// Mitsubishi GX Works2 project: plc0806   PLC: Q03UDV

PROGRAM MAIN
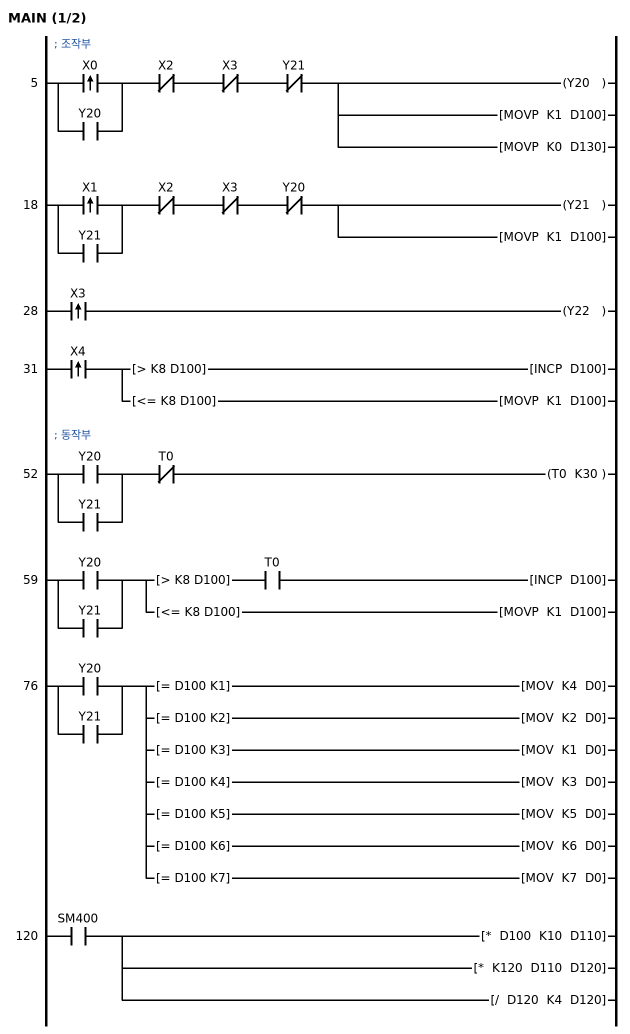
; 조작부
5     LDP     X0
      OR      Y20
      ANI     X2
      ANI     X3
      ANI     Y21
      OUT     Y20
      MOVP    K1 D100
      MOVP    K0 D130
18    LDP     X1
      OR      Y21
      ANI     X2
      ANI     X3
      ANI     Y20
      OUT     Y21
      MOVP    K1 D100
28    LDP     X3
      OUT     Y22
31    LDP     X4
      MPS
      AND>    K8 D100
      INCP    D100
      MPP
      AND<=   K8 D100
      MOVP    K1 D100
; 동작부
52    LD      Y20
      OR      Y21
      ANI     T0
      OUT     T0 K30
59    LD      Y20
      OR      Y21
      MPS
      AND>    K8 D100
      AND     T0
      INCP    D100
      MPP
      AND<=   K8 D100
      MOVP    K1 D100
76    LD      Y20
      OR      Y21
      MPS
      AND=    D100 K1
      MOV     K4 D0
      MRD
      AND=    D100 K2
      MOV     K2 D0
      MRD
      AND=    D100 K3
      MOV     K1 D0
      MRD
      AND=    D100 K4
      MOV     K3 D0
      MRD
      AND=    D100 K5
      MOV     K5 D0
      MRD
      AND=    D100 K6
      MOV     K6 D0
      MPP
      AND=    D100 K7
      MOV     K7 D0
120   LD      SM400
      *       D100 K10 D110
      *       K120 D110 D120
      /       D120 K4 D120
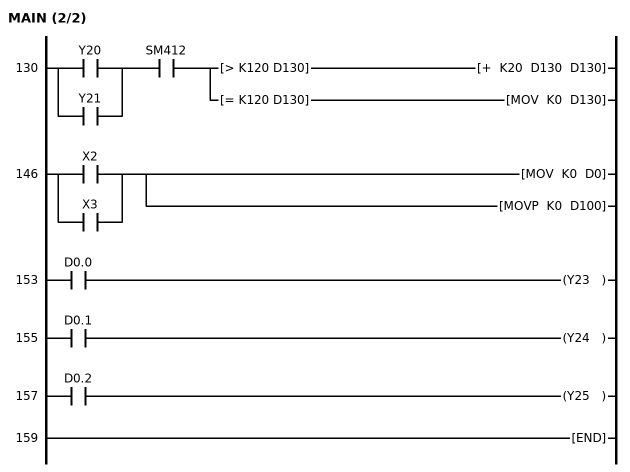
130   LD      Y20
      OR      Y21
      AND     SM412
      MPS
      AND>    K120 D130
      +       K20 D130 D130
      MPP
      AND=    K120 D130
      MOV     K0 D130
146   LD      X2
      OR      X3
      MOV     K0 D0
      MOVP    K0 D100
153   LD      D0.0
      OUT     Y23
155   LD      D0.1
      OUT     Y24
157   LD      D0.2
      OUT     Y25
159   END
END_PROGRAM

PROGRAM laundry
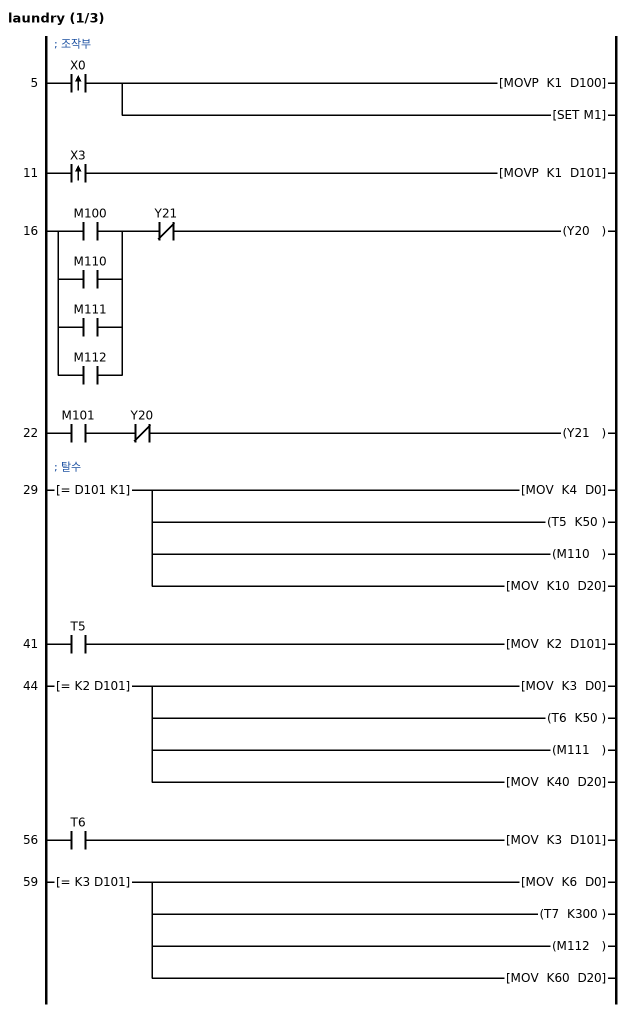
; 조작부
5     LDP     X0
      MOVP    K1 D100
      SET     M1
11    LDP     X3
      MOVP    K1 D101
16    LD      M100
      OR      M110
      OR      M111
      OR      M112
      ANI     Y21
      OUT     Y20
22    LD      M101
      ANI     Y20
      OUT     Y21
; 탈수
29    LD=     D101 K1
      MOV     K4 D0
      OUT     T5 K50
      OUT     M110
      MOV     K10 D20
41    LD      T5
      MOV     K2 D101
44    LD=     K2 D101
      MOV     K3 D0
      OUT     T6 K50
      OUT     M111
      MOV     K40 D20
56    LD      T6
      MOV     K3 D101
59    LD=     K3 D101
      MOV     K6 D0
      OUT     T7 K300
      OUT     M112
      MOV     K60 D20
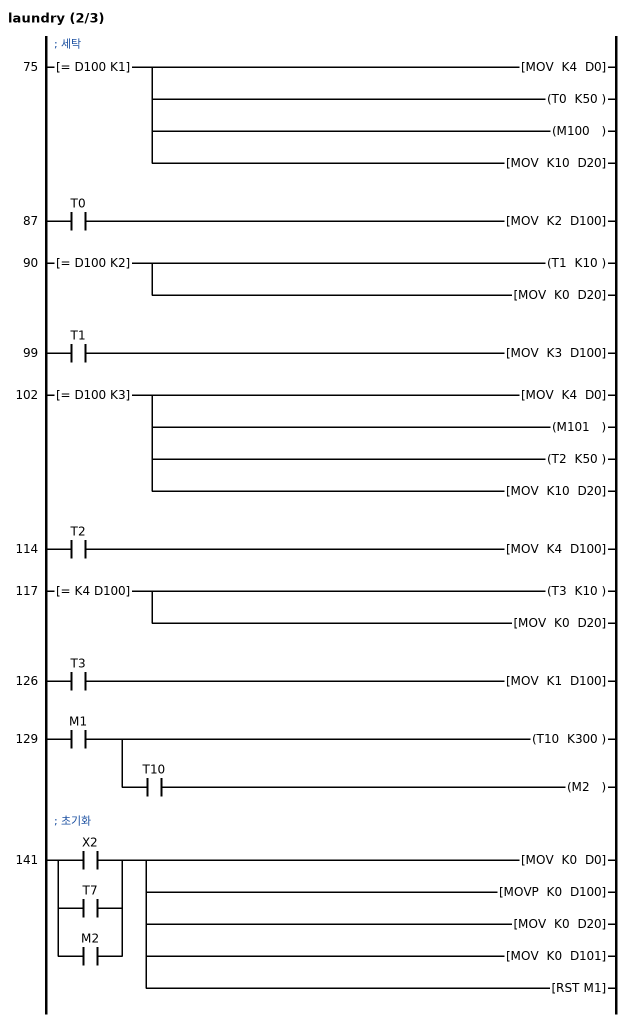
; 세탁
75    LD=     D100 K1
      MOV     K4 D0
      OUT     T0 K50
      OUT     M100
      MOV     K10 D20
87    LD      T0
      MOV     K2 D100
90    LD=     D100 K2
      OUT     T1 K10
      MOV     K0 D20
99    LD      T1
      MOV     K3 D100
102   LD=     D100 K3
      MOV     K4 D0
      OUT     M101
      OUT     T2 K50
      MOV     K10 D20
114   LD      T2
      MOV     K4 D100
117   LD=     K4 D100
      OUT     T3 K10
      MOV     K0 D20
126   LD      T3
      MOV     K1 D100
129   LD      M1
      OUT     T10 K300
      AND     T10
      OUT     M2
; 초기화
141   LD      X2
      OR      T7
      OR      M2
      MOV     K0 D0
      MOVP    K0 D100
      MOV     K0 D20
      MOV     K0 D101
      RST     M1
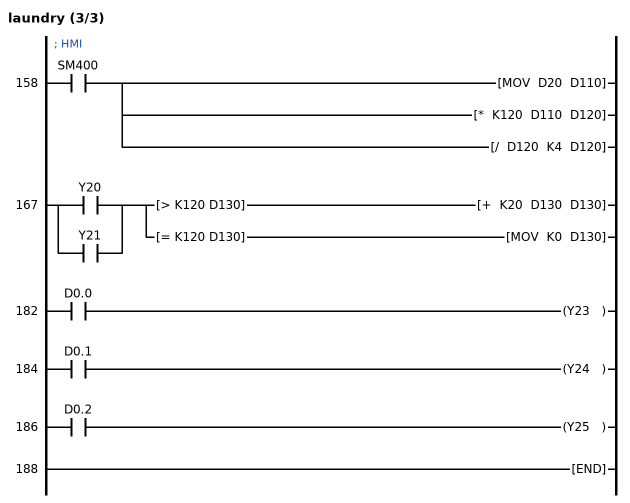
; HMI
158   LD      SM400
      MOV     D20 D110
      *       K120 D110 D120
      /       D120 K4 D120
167   LD      Y20
      OR      Y21
      MPS
      AND>    K120 D130
      +       K20 D130 D130
      MPP
      AND=    K120 D130
      MOV     K0 D130
182   LD      D0.0
      OUT     Y23
184   LD      D0.1
      OUT     Y24
186   LD      D0.2
      OUT     Y25
188   END
END_PROGRAM
